TYPE ST_ProductDataA :
STRUCT
	nQuality : UINT;
	bGoodProduct : BOOL;
END_STRUCT
END_TYPE

(* stored: Version 1.1.0.1, ProductVersion 3.1.4024.12
   DUT ST_ProductDataA: Id {2901f777-4d1f-4c61-8edd-19521f1bfbbb} *)
